FUNCTION F_DWORD_ARG : ST_Arg
VAR_INPUT
	dwInput : DWORD;
END_VAR
VAR
	stArg : ST_Arg;
	sysVar_Info : __SYSTEM.VAR_INFO;
END_VAR

sysVar_Info 	:= __VARINFO(dwInput);
stArg.TypeClass := sysVar_Info.TypeClass;
stArg.pValue 	:= 0;
stArg.diSize 	:= SIZEOF(dwInput);
stArg.sValue 	:= TO_STRING(dwInput); 
F_DWORD_ARG := stArg;

END_FUNCTION

(* stored: Version 1.1.0.1, ProductVersion 3.1.4024.4
   POU F_DWORD_ARG: Id {da34ecc2-db0e-4cee-9f11-22bc92f03260}, SpecialFunc None *)
